PROGRAM SturingVerwarming
VAR
	fbGroteVergaderzaal					:fbVerwarming;
	fbKleineVergaderzaal				:fbVerwarming;
	fbBureau							:fbVerwarming;
	
	bDrukknopGroteZaal			AT %I*		:BOOL; //Drukknoppen te voorzien op kast
	bDrukknopKleineZaal			AT %I*		:BOOL; //Drukknoppen te voorzien op kast
	bDrukknopBureau				AT %I*		:BOOL; //Drukknoppen te voorzien op kast
	
	bThermostaatGroteZaal		AT %I*		:BOOL; 
	bThermostaatKleineZaal		AT %I*		:BOOL;
	bThermostaatBureau			AT %I*		:BOOL;
	
	bKlepGroteZaal				AT %Q*		:BOOL; 	//Uitgangen naar relais in kastje aan brander
	bKlepKleineZaal				AT %Q*		:BOOL; 	//Uitgangen naar relais in kastje aan brander
	bKlepBureau					AT %Q*		:BOOL;	//Uitgangen naar relais in kastje aan brander
	bBranderAan					AT %Q*		:BOOL; 	//Uitgangen naar relais in kastje aan brander
	bKlepKleineZaalLamp			AT %Q*		:BOOL; 	//Uitgangen naar lamp in hoofdkast
	bKlepBureauLamp				AT %Q*		:BOOL;	//Uitgangen naar lamp in hoofdkast
	bKlepGroteZaalLamp				AT %Q*		:BOOL; 	//Uitgangen naar lamp in hoofdkast
	
	bLichtReactief							:BOOL := FALSE;
	tLoopTijdVerwarming 					:TIME := T#4H; 
	
	// tTijdVoorStart is de tijd dat de verwarming aangaat nadat iemand op de knop druk, die op de kast voorzien is.
	
END_VAR

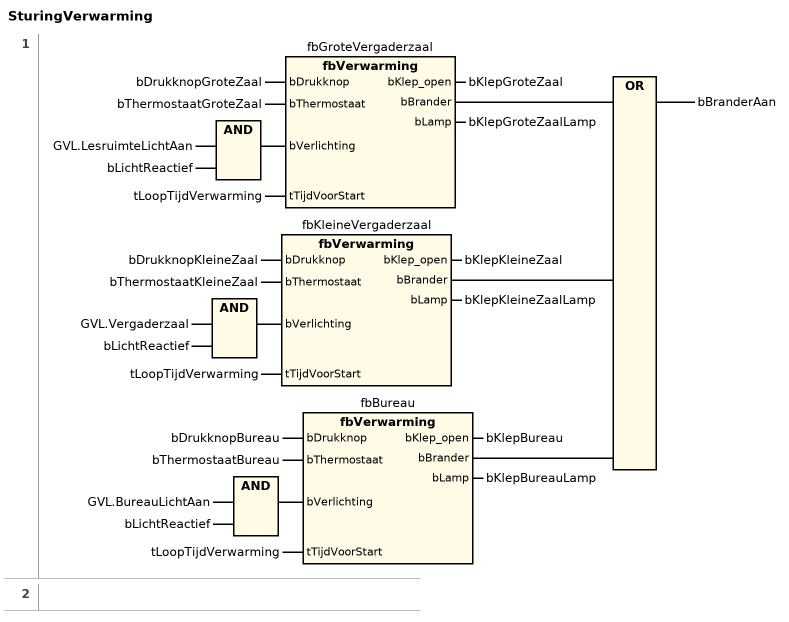
// NETWORK 1
fbGroteVergaderzaal(
    bDrukknop := bDrukknopGroteZaal,
    bThermostaat := bThermostaatGroteZaal,
    bVerlichting := GVL.LesruimteLichtAan AND bLichtReactief,
    tTijdVoorStart := tLoopTijdVerwarming,
    bKlep_open => bKlepGroteZaal,
    bLamp => bKlepGroteZaalLamp); // fbVerwarming
fbKleineVergaderzaal(
    bDrukknop := bDrukknopKleineZaal,
    bThermostaat := bThermostaatKleineZaal,
    bVerlichting := GVL.Vergaderzaal AND bLichtReactief,
    tTijdVoorStart := tLoopTijdVerwarming,
    bKlep_open => bKlepKleineZaal,
    bLamp => bKlepKleineZaalLamp); // fbVerwarming
fbBureau(
    bDrukknop := bDrukknopBureau,
    bThermostaat := bThermostaatBureau,
    bVerlichting := GVL.BureauLichtAan AND bLichtReactief,
    tTijdVoorStart := tLoopTijdVerwarming,
    bKlep_open => bKlepBureau,
    bLamp => bKlepBureauLamp); // fbVerwarming
bBranderAan := fbGroteVergaderzaal.bBrander OR fbKleineVergaderzaal.bBrander OR fbBureau.bBrander;

// NETWORK 2

END_PROGRAM

(* stored: Version 1.1.0.1, ProductVersion 3.1.4024.12
   POU SturingVerwarming: Id {07ea3488-9e2d-4cf5-9f83-ee7835ac8045}, SpecialFunc None *)
